FUNCTION_BLOCK ServiceCylinder
VAR_INPUT
	ptBlock : POINTER TO CylinderBlockBase;
END_VAR
VAR_OUTPUT
END_VAR
VAR
	nCounter : WORD := 0;
	bMatched : BOOL := false;
	
	tmrWatchDog: TON;
END_VAR

//Run timers
ptBlock^.TMR_WATCH_DOG(IN:= , PT:= , Q=> , ET=> );
ptBlock^.TMR_DELAY_TO_A(IN:= , PT:= , Q=> , ET=> );
ptBlock^.TMR_DELAY_TO_B(IN:= , PT:= , Q=> , ET=> );

// scan all sensor status
ptBlock^.BIT_A_MATCH := TRUE;
FOR nCounter := 1 TO ptBlock^.A_SENSOR_USED_COUNT BY 1 DO
	ptBlock^.BIT_A_MATCH := (ptBlock^.BIT_A_MATCH AND ptBlock^.SENSOR_A[nCounter]);
END_FOR
ptBlock^.BIT_B_MATCH := TRUE;
FOR nCounter := 1 TO ptBlock^.B_SENSOR_USED_COUNT BY 1 DO
	ptBlock^.BIT_B_MATCH := (ptBlock^.BIT_B_MATCH AND ptBlock^.SENSOR_B[nCounter]);
END_FOR

// if watch dog had been reset due to command changed in previous scan
// restart
IF NOT ptBlock^.TMR_WATCH_DOG.IN THEN
	ptBlock^.TMR_WATCH_DOG.IN := TRUE;
END_IF

// once command changes , reset timer counter
IF ptBlock^.COMMAND_CACHED <> ptBlock^.LAST_COMMAND THEN
	//ptBlock^.TMR_WATCH_DOG.IN:=false;	//invalid , do not across a scan
	ptBlock^.TMR_WATCH_DOG.IN:=FALSE;
	ptBlock^.TMR_DELAY_TO_A.IN := (ptBlock^.COMMAND_CACHED=eCylinderCommands.COMMAND_A); //active A delay timer
	ptBlock^.TMR_DELAY_TO_B.IN := (ptBlock^.COMMAND_CACHED=eCylinderCommands.COMMAND_B); //if no sensor B , active B delay timer
	
	//reset done/warn
	ptBlock^.BIT_DONE := FALSE;
	ptBlock^.BIT_WARNING := FALSE;
	
	//output process
	FOR nCounter:=1 TO 2 BY 1 DO
		ptBlock^.ACT_A[nCounter] := (ptBlock^.COMMAND_CACHED = eCylinderCommands.COMMAND_A);
		ptBlock^.ACT_B[nCounter] := (ptBlock^.COMMAND_CACHED = eCylinderCommands.COMMAND_B);
	END_FOR
	
END_IF


//reset
bMatched := FALSE;
// Check if match
CASE ptBlock^.COMMAND_CACHED OF
	eCylinderCommands.NO_COMMAND:
	bMatched:= TRUE;
	
	eCylinderCommands.COMMAND_A:
	IF ptBlock^.TMR_DELAY_TO_A.Q THEN
		bMatched:= (ptBlock^.BIT_A_MATCH ) AND (NOT ptBlock^.BIT_B_MATCH OR ptBlock^.B_SENSOR_USED_COUNT=0);
	END_IF
	
	eCylinderCommands.COMMAND_B:
	IF ptBlock^.TMR_DELAY_TO_B.Q THEN
		bMatched:= (NOT ptBlock^.BIT_A_MATCH OR ptBlock^.A_SENSOR_USED_COUNT=0) AND (ptBlock^.BIT_B_MATCH );
	END_IF
		
END_CASE

// status update
ptBlock^.BIT_DONE := bMatched OR (NOT bMatched AND ptBlock^.BIT_WARN_SUPPRESS AND ptBlock^.TMR_WATCH_DOG.Q);
ptBlock^.BIT_WARNING := NOT bMatched AND NOT ptBlock^.BIT_WARN_SUPPRESS AND ptBlock^.TMR_WATCH_DOG.Q;


// cache last command
ptBlock^.LAST_COMMAND := ptBlock^.COMMAND_CACHED;

END_FUNCTION_BLOCK

(* stored: Version 1.1.0.1, ProductVersion 3.1.4020.12
   POU ServiceCylinder: Id {a99bf5d1-aaa3-4095-9742-005d9ab3fed8}, SpecialFunc None *)
